# EPICS StreamDevice protocol: pmacUtilApp/protocol/encoderRead.proto
Terminator = CR;
InTerminator = CR "\x06";

LockTimeout = 10000;
ReplyTimeout = 500;
ReadTimeout = 500;

getPos {
    out "#\$1 P"; in "%f";
}
